INTERFACE I_FallibleUsint


PROPERTY Error : BOOL
GET
END_GET
END_PROPERTY


PROPERTY Value : USINT
GET
END_GET
END_PROPERTY

END_INTERFACE

(* stored: Version 1.1.0.1
   Itf I_FallibleUsint: Id {a1b2c3d4-0004-4001-8001-000000000031}
   Property Error: Id {a1b2c3d4-0004-4001-8001-000000000032}
   Get Get: Id {a1b2c3d4-0004-4001-8001-000000000033}
   Property Value: Id {a1b2c3d4-0004-4001-8001-000000000034}
   Get Get: Id {a1b2c3d4-0004-4001-8001-000000000035} *)
